FUNCTION_BLOCK E_MERGE_6 (* Composite Function Block Type *)
  (* Standard: 61499-2 *)
  (* Version 0.0, 2018-11-02, 4DIAC-IDE, 4DIAC-Consortium *)
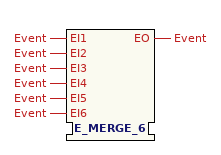
  EVENT_INPUT
    EI1;
    EI2;
    EI3;
    EI4;
    EI5;
    EI6;
  END_EVENT
  EVENT_OUTPUT
    EO;
  END_EVENT
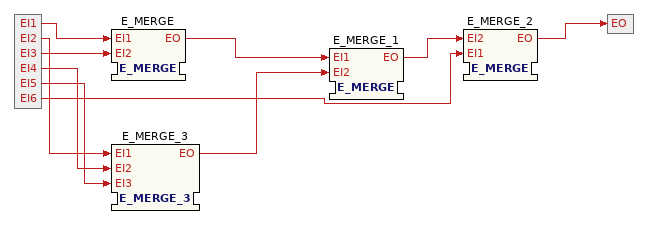
  FBS
    E_MERGE : E_MERGE;
    E_MERGE_3 : E_MERGE_3;
    E_MERGE_1 : E_MERGE;
    E_MERGE_2 : E_MERGE;
  END_FBS
  EVENT_CONNECTIONS
    EI1 TO E_MERGE.EI1;
    EI2 TO E_MERGE.EI2;
    EI3 TO E_MERGE_3.EI1;
    EI4 TO E_MERGE_3.EI2;
    EI5 TO E_MERGE_3.EI3;
    E_MERGE.EO TO E_MERGE_1.EI1;
    E_MERGE_3.EO TO E_MERGE_1.EI2;
    E_MERGE_1.EO TO E_MERGE_2.EI2;
    EI6 TO E_MERGE_2.EI1;
    E_MERGE_2.EO TO EO;
  END_CONNECTIONS
END_FUNCTION_BLOCK
